// TIA Portal V16 export
// export: Created 2026-06-22T01:28:19.1806514Z, ExportSetting WithDefaults, DisplayName Totally Integrated Automation Portal, DisplayVersion V16 Update 8, DisplayName TIA Portal Version Control Interface, DisplayVersion V16 Update 8, DisplayName TIA Portal Openness, DisplayVersion V16 Update 8, DisplayName SINAMICS Startdrive Advanced, DisplayVersion V16, DisplayName SINAMICS Startdrive G130, G150, S120, S150, SINAMICS MV, S210, DisplayVersion V16, DisplayName SINAMICS Startdrive G110M, G120, G120C, G120D, G120P, DisplayVersion V16, DisplayName STEP 7 Professional, DisplayVersion V16 Update 8, DisplayName STEP 7 Safety, DisplayVersion V16 Update 7, DisplayName WinCC Advanced, DisplayVersion V16 Update 8
TagTable "默认变量表"
  Tag_ScreenNumber : UInt  (1 s)
  Button : Bool  (1 s)
  Light : Bool  (1 s)
  BTN_Motor_Start : Bool  (1 s)
  BTN_Motor_Stop : Bool  (1 s)
  BTN_Motor_Reset : Bool  (1 s)
  STS_Motor_Running : Bool  (1 s)
  LMP_Motor_Fault : Bool  (1 s)
  IO_Motor_Speed : Int  (1 s)
  SIO_Motor_Mode : Int  (1 s)
